// TIA Portal V19 export
TYPE "dtStepCond"
   STRUCT
      count : Bool;   // TRUE: The conditional timer should start counting the preset duration (types 0, 2)
      reset : Bool;   // TRUE: The conditional timer should reset (types 0, 2)
      proceed : Bool;   // TRUE: The step should end and proceed to next (types 1,2)
      prompt : Bool;   // TRUE: The step is requesting a prompt for confirmation
      nofault : Bool;   // TRUE: There is no critical fault for this step
   END_STRUCT;
END_TYPE
